PROGRAM Exec_ISO
VAR
	FB_exe_ISO:FB_Exec_ISO3_libTC3_V2;	
	ItpWriteRParams_1:ItpWriteRParamsex;
	B_Reset:BOOL;	
	FB_WriteGrpMinVeloTrans_1: FB_WriteGrpMinVeloTrans;
	FB_WriteGrpMinVeloTrans_error: BOOL;
	
	GetRParam	:ItpReadRParamsEx;
	 TON_ReadRParam	:TON;
	 R5_FromNciToPlc	:LREAL;
END_VAR

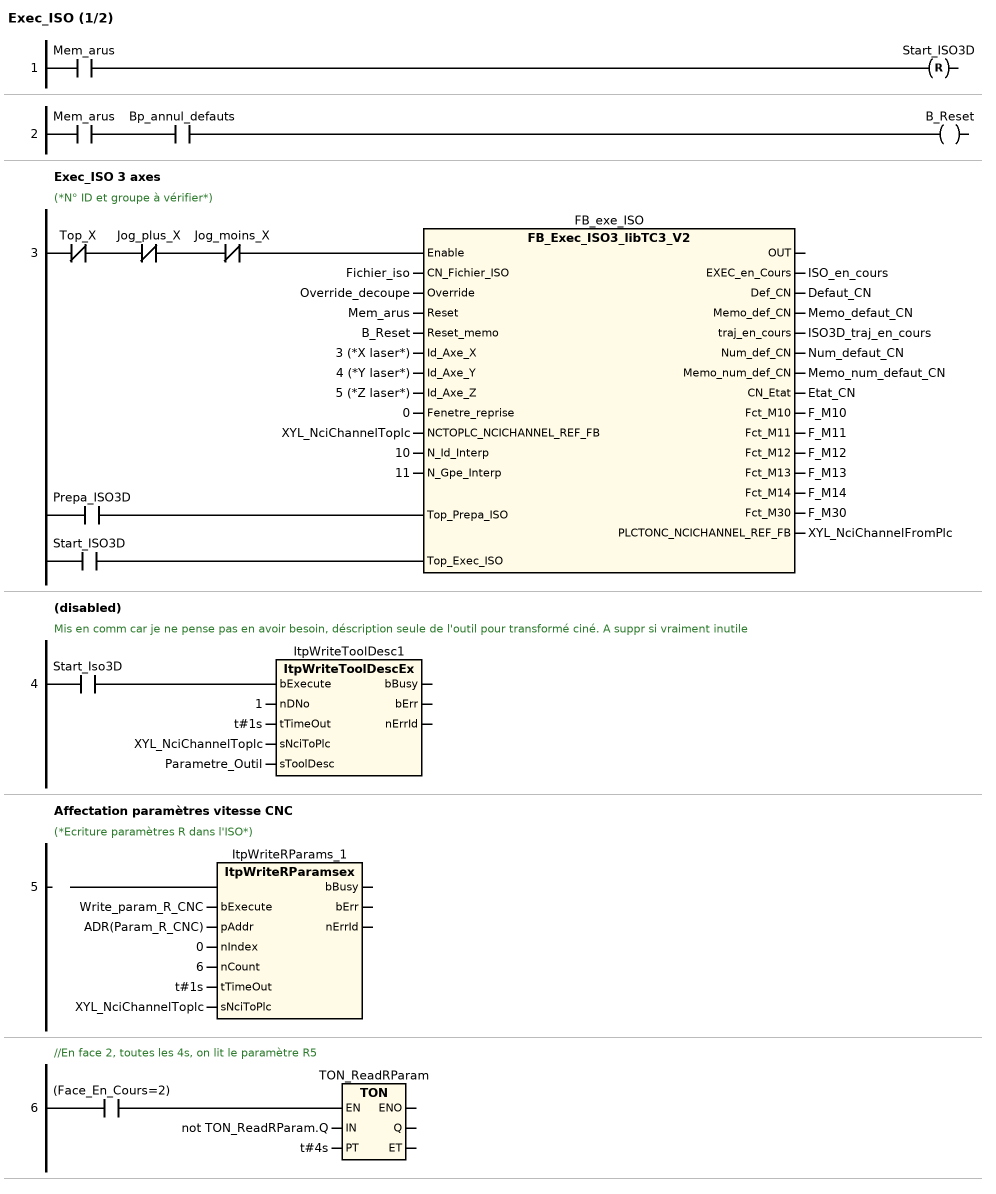
// NETWORK 1
Start_ISO3D R= Mem_arus;

// NETWORK 2
B_Reset := Mem_arus AND Bp_annul_defauts;

// NETWORK 3: Exec_ISO 3 axes
// (*N° ID et groupe à vérifier*)
FB_exe_ISO(
    Enable := NOT Top_X AND NOT Jog_plus_X AND NOT Jog_moins_X,
    CN_Fichier_ISO := Fichier_iso,
    Override := Override_decoupe,
    Reset := Mem_arus,
    Reset_memo := B_Reset,
    Id_Axe_X := 3 (*X laser*),
    Id_Axe_Y := 4 (*Y laser*),
    Id_Axe_Z := 5 (*Z laser*),
    Fenetre_reprise := 0,
    NCTOPLC_NCICHANNEL_REF_FB := XYL_NciChannelToplc,
    N_Id_Interp := 10,
    N_Gpe_Interp := 11,
    Top_Prepa_ISO := Prepa_ISO3D,
    Top_Exec_ISO := Start_ISO3D,
    EXEC_en_Cours => ISO_en_cours,
    Def_CN => Defaut_CN,
    Memo_def_CN => Memo_defaut_CN,
    traj_en_cours => ISO3D_traj_en_cours,
    Num_def_CN => Num_defaut_CN,
    Memo_num_def_CN => Memo_num_defaut_CN,
    CN_Etat => Etat_CN,
    Fct_M10 => F_M10,
    Fct_M11 => F_M11,
    Fct_M12 => F_M12,
    Fct_M13 => F_M13,
    Fct_M14 => F_M14,
    Fct_M30 => F_M30,
    PLCTONC_NCICHANNEL_REF_FB => XYL_NciChannelFromPlc); // FB_Exec_ISO3_libTC3_V2

// NETWORK 4 (disabled)
// Mis en comm car je ne pense pas en avoir besoin, déscription seule de l'outil pour transformé ciné. A suppr si vraiment inutile
// ItpWriteToolDesc1(
//     bExecute := Start_Iso3D,
//     nDNo := 1,
//     tTimeOut := t#1s,
//     sNciToPlc := XYL_NciChannelToplc,
//     sToolDesc := Parametre_Outil); // ItpWriteToolDescEx

// NETWORK 5: Affectation paramètres vitesse CNC
// (*Ecriture paramètres R dans l'ISO*)
ItpWriteRParams_1(
    bExecute := Write_param_R_CNC,
    pAddr := ADR(Param_R_CNC),
    nIndex := 0,
    nCount := 6,
    tTimeOut := t#1s,
    sNciToPlc := XYL_NciChannelToplc); // ItpWriteRParamsex

// NETWORK 6
// //En face 2, toutes les 4s, on lit le paramètre R5
IF (Face_En_Cours=2) THEN
    TON_ReadRParam(IN := not TON_ReadRParam.Q, PT := t#4s); // TON
END_IF

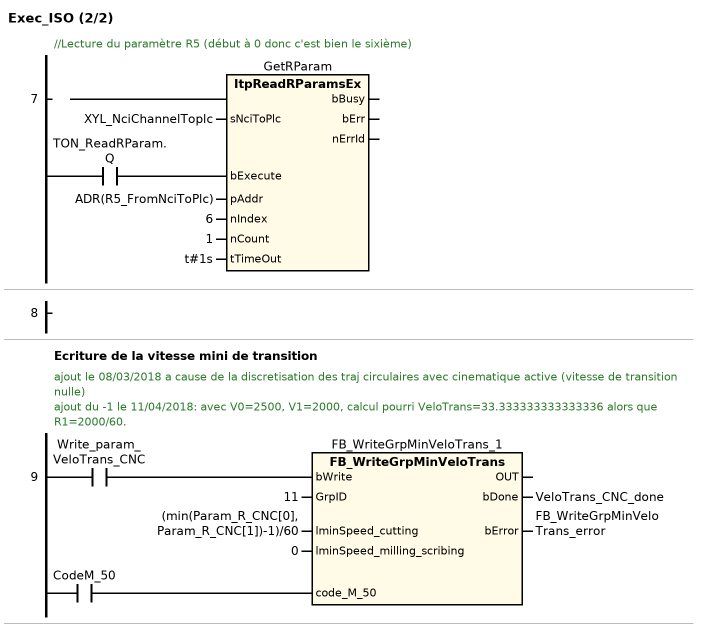
// NETWORK 7
// //Lecture du paramètre R5 (début à 0 donc c'est bien le sixième)
GetRParam(
    sNciToPlc := XYL_NciChannelToplc,
    bExecute := TON_ReadRParam.Q,
    pAddr := ADR(R5_FromNciToPlc),
    nIndex := 6,
    nCount := 1,
    tTimeOut := t#1s); // ItpReadRParamsEx

// NETWORK 8

// NETWORK 9: Ecriture de la vitesse mini de transition
// ajout le 08/03/2018 a cause de la discretisation des traj circulaires avec cinematique active (vitesse de transition nulle)
// ajout du -1 le 11/04/2018: avec V0=2500, V1=2000, calcul pourri VeloTrans=33.333333333333336 alors que R1=2000/60.
FB_WriteGrpMinVeloTrans_1(
    bWrite := Write_param_VeloTrans_CNC,
    GrpID := 11,
    lminSpeed_cutting := (min(Param_R_CNC[0],Param_R_CNC[1])-1)/60,
    lminSpeed_milling_scribing := 0,
    code_M_50 := CodeM_50,
    bDone => VeloTrans_CNC_done,
    bError => FB_WriteGrpMinVeloTrans_error); // FB_WriteGrpMinVeloTrans

END_PROGRAM

(* stored: Version 1.1.0.1, ProductVersion 3.1.4024.15
   POU Exec_ISO: Id {8e785ce0-df6d-4c42-83ab-89667263c0ee}, SpecialFunc None *)
